PROGRAM PRG_1_PlcTask
VAR

END_VAR

PRG_MR1L0_HOMS_States();
PRG_MR2L0_HOMS_States();
PRG_PMPS();

END_PROGRAM

(* stored: Version 1.1.0.1, ProductVersion 3.1.4022.18
   POU PRG_1_PlcTask: Id {6c74c1b3-089b-4af5-bdef-e72814f71ef8}, SpecialFunc None *)
